// TwinCAT 3 PLC project _4_sequence_automatique
// ProgramVersion: 3.1.4020.2
// libraries:
//   Tc2_Standard, * (Beckhoff Automation GmbH)
//   Tc2_System, * (Beckhoff Automation GmbH)
//   Tc3_Module, * (Beckhoff Automation GmbH)
// project tree:
//   / PlcTask.TcTTO
//   POUs/ MAIN.TcPOU
// (motion and I/O tree: see PLC project 1calcul)
// real-time tasks:
//   TASK PlcTask: cycle T#1ms, priority 20, ADS port 350
// variable links:

CONFIGURATION _4_sequence_automatique
    RESOURCE PLC ON TwinCAT3
        TASK PlcTask(INTERVAL := T#10ms, PRIORITY := 20);
        PROGRAM MAIN WITH PlcTask : MAIN;
    END_RESOURCE
END_CONFIGURATION

// ---- POUs/MAIN.TcPOU
PROGRAM MAIN
VAR
	iStep: INT :=0; //etape
END_VAR
VAR_INPUT
	IxFdcSort, IxFdcRentree: BOOL :=0; //fin de course verin | avec AT %I si lien physique
END_VAR
VAR_OUTPUT
	QxFdcSort, QxFdcRentree: BOOL := 0; //actionner le verin | avec AT %Q si lien physique
END_VAR

CASE iStep OF
	0: iStep:=100;
	100: //sortir verin et attendre le FDC
		IF IxFdcSort THEN
			IxFdcSort:=FALSE; //options simulateur
			iStep:=200;
		END_IF
	200: //rentrer le verin
		IF IxFdcRentree THEN
			IxFdcRentree:=FALSE; //options simulation
			iStep:=100;
		END_IF
END_CASE

//Actions
QxFdcRentree:=iStep=200;
QxFdcSort:=iStep=100;

END_PROGRAM
